// Mitsubishi GX Works2 project: 2. bsfl   PLC: Q03UDV

PROGRAM MAIN
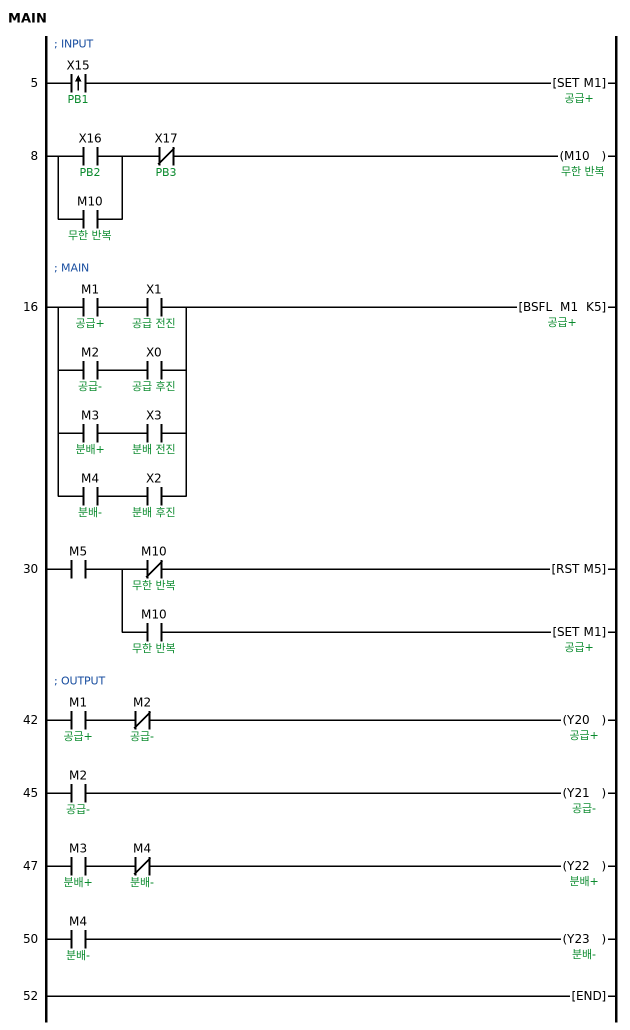
; INPUT
5     LDP     X15  ; PB1
      SET     M1  ; 공급+
8     LD      X16  ; PB2
      OR      M10  ; 무한 반복
      ANI     X17  ; PB3
      OUT     M10  ; 무한 반복
; MAIN
16    LD      M1  ; 공급+
      AND     X1  ; 공급 전진
      LD      M2  ; 공급-
      AND     X0  ; 공급 후진
      ORB
      LD      M3  ; 분배+
      AND     X3  ; 분배 전진
      ORB
      LD      M4  ; 분배-
      AND     X2  ; 분배 후진
      ORB
      BSFL    M1 K5
30    LD      M5
      MPS
      ANI     M10  ; 무한 반복
      RST     M5
      MPP
      AND     M10  ; 무한 반복
      SET     M1  ; 공급+
; OUTPUT
42    LD      M1  ; 공급+
      ANI     M2  ; 공급-
      OUT     Y20  ; 공급+
45    LD      M2  ; 공급-
      OUT     Y21  ; 공급-
47    LD      M3  ; 분배+
      ANI     M4  ; 분배-
      OUT     Y22  ; 분배+
50    LD      M4  ; 분배-
      OUT     Y23  ; 분배-
52    END
END_PROGRAM

// device comments not shown above
X4  ; 가공 상승
X1C  ; Toggle
P1  ; STOP
